(* Logix 5000 project; controller APM Emulate 5570 rev 30.12; software revision 30.00 *)

TASK MainTask (continuous, watchdog 500 ms) : MainProgram

MODULES
   Local : Emulate 5570 (ICP 2, rev 30.12)
      I_O1 : vendor 1 type 0 code 15 (ICP 3, rev 1.1, Output RPI 150 ms)
      I_O2 : vendor 1 type 0 code 15 (ICP 4, rev 1.1, Output RPI 150 ms)
END_MODULES

VAR_GLOBAL   (* controller tags *)
   CT_AXIS_DIST : AXIS_VIRTUAL;
   MTN : MOTION_GROUP;
   PNT_AXIS_MTA : AXIS_VIRTUAL;
   PNT_AXIS_MTB : AXIS_VIRTUAL;
   PNT_AXIS_MTC : AXIS_VIRTUAL;
END_VAR

PROGRAM MainProgram   (* main routine MainRoutine *)
VAR
   CT_ACT_CT0 : BOOL;
   CT_ACT_CT1 : BOOL;
   CT_ACT_CT2 : BOOL;
   CT_ACT_CT3 : BOOL;
   CT_ACT_CT4 : BOOL;
   CT_ACT_CT5 : BOOL;
   CT_ACT_CT6 : BOOL;
   CT_ACT_HOM0 : BOOL;
   CT_ACT_HOM1 : BOOL;
   CT_ACT_HOM2 : BOOL;
   CT_ACT_HOM3 : BOOL;
   CT_ACT_STP : BOOL;
   CT_AXIS_CT1 : MOTION_INSTRUCTION;
   CT_AXIS_CT4 : MOTION_INSTRUCTION;
   CT_AXIS_HOM0 : MOTION_INSTRUCTION;
   CT_AXIS_HOM1 : MOTION_INSTRUCTION;
   CT_AXIS_HOM2 : MOTION_INSTRUCTION;
   CT_CA_AVC : BOOL;
   CT_CA_RET : BOOL;
   CT_CC_AVC : BOOL;
   CT_CC_RET : BOOL;
   CT_CNT1 : COUNTER := (PRE := 18);
   CT_CP_AVC : BOOL;
   CT_CP_RET : BOOL;
   CT_DIST : INT;
   CT_ISOVER : BOOL;
   CT_MASD_DIST : MOTION_INSTRUCTION;
   CT_MASR_DIST : MOTION_INSTRUCTION;
   CT_OK : BOOL;
   CT_PBT_ESTP : ALIAS FOR Local:4:I.Data[1].0;
   CT_PBT_HOM : ALIAS FOR Local:4:I.Data[1].2;
   CT_PBT_STA : ALIAS FOR Local:4:I.Data[1].1;
   CT_SEN_CaAvc : ALIAS FOR Local:4:I.Data[1].4;
   CT_SEN_CaRet : ALIAS FOR Local:4:I.Data[1].3;
   CT_SEN_CcAvc : ALIAS FOR Local:4:I.Data[1].6;
   CT_SEN_CcRet : ALIAS FOR Local:4:I.Data[1].5;
   CT_SEN_CpAvc : ALIAS FOR Local:4:I.Data[1].8;
   CT_SEN_CpRet : ALIAS FOR Local:4:I.Data[1].7;
   CT_SEN_MAT : ALIAS FOR Local:4:I.Data[1].9;
   MAIN_ACTIVE : BOOL;
   MAIN_PBT_ESTP : ALIAS FOR Local:3:I.Data[1].0;
   MAIN_PBT_STA : ALIAS FOR Local:3:I.Data[1].1;
   PNT_ACT1_MTA_MAM : MOTION_INSTRUCTION;
   PNT_ACT1_MTB_MAM : MOTION_INSTRUCTION;
   PNT_ACT2_MTC_MAM : MOTION_INSTRUCTION;
   PNT_ACT3_MTA_MAM : MOTION_INSTRUCTION;
   PNT_ACT3_MTB_MAM : MOTION_INSTRUCTION;
   PNT_ACT_0 : BOOL;
   PNT_ACT_1 : BOOL;
   PNT_ACT_2 : BOOL;
   PNT_ACT_3 : BOOL;
   PNT_ACT_4 : BOOL;
   PNT_ACT_HOM : BOOL;
   PNT_ACTH_MTA_MAM : MOTION_INSTRUCTION;
   PNT_ACTH_MTB_MAM : MOTION_INSTRUCTION;
   PNT_ACTH_MTC_MAM : MOTION_INSTRUCTION;
   PNT_CNT1 : COUNTER := (PRE := 3);
   PNT_ISHOM : BOOL;
   PNT_ISOVER : BOOL;
   PNT_MASD_MTA : MOTION_INSTRUCTION;
   PNT_MASD_MTB : MOTION_INSTRUCTION;
   PNT_MASD_MTC : MOTION_INSTRUCTION;
   PNT_MASR_MTA : MOTION_INSTRUCTION;
   PNT_MASR_MTB : MOTION_INSTRUCTION;
   PNT_MASR_MTC : MOTION_INSTRUCTION;
   PNT_MTA_AVC : BOOL;
   PNT_MTA_RET : BOOL;
   PNT_MTA_STP : BOOL;
   PNT_MTB_AVC : BOOL;
   PNT_MTB_RET : BOOL;
   PNT_MTB_STP : BOOL;
   PNT_MTC_AVC : BOOL;
   PNT_MTC_RET : BOOL;
   PNT_MTC_STP : BOOL;
   PNT_PBT_HOM : ALIAS FOR Local:3:I.Data[1].10;
   PNT_PBT_STA : ALIAS FOR Local:3:I.Data[1].11;
   PNT_PBT_STP : ALIAS FOR Local:3:I.Data[1].12;
   PNT_SEN_1 : ALIAS FOR Local:3:I.Data[1].13;
   PNT_SEN_2 : ALIAS FOR Local:3:I.Data[1].14;
   PNT_SEN_3 : ALIAS FOR Local:3:I.Data[1].15;
   PNT_SEN_4 : ALIAS FOR Local:3:I.Data[1].16;
   PNT_SEN_5 : ALIAS FOR Local:3:I.Data[1].17;
   PNT_SEN_6 : ALIAS FOR Local:3:I.Data[1].18;
   PNT_SEN_7 : ALIAS FOR Local:3:I.Data[1].19;
   PNT_TM1 : TIMER := (PRE := 2000);
END_VAR

ROUTINE Corte_actions   (* ladder *)
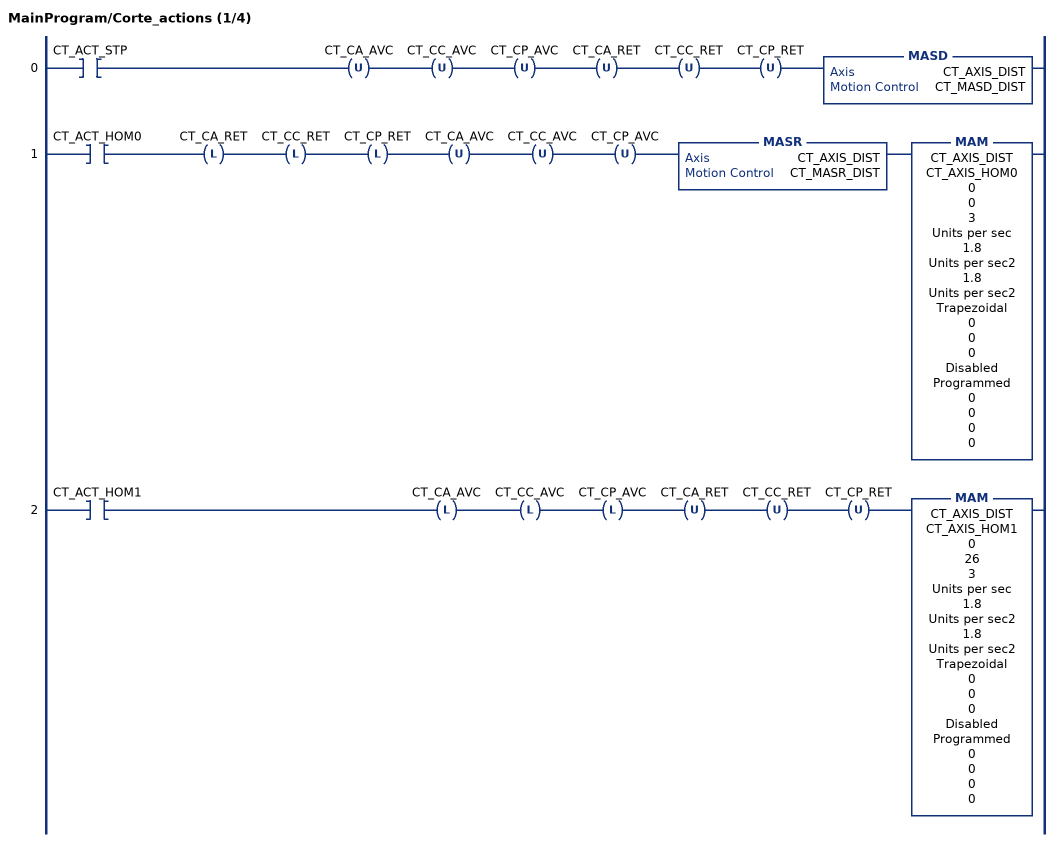
   0: XIC(CT_ACT_STP)OTU(CT_CA_AVC)OTU(CT_CC_AVC)OTU(CT_CP_AVC)OTU(CT_CA_RET)OTU(CT_CC_RET)OTU(CT_CP_RET)MASD(CT_AXIS_DIST,CT_MASD_DIST);
   1: XIC(CT_ACT_HOM0)OTL(CT_CA_RET)OTL(CT_CC_RET)OTL(CT_CP_RET)OTU(CT_CA_AVC)OTU(CT_CC_AVC)OTU(CT_CP_AVC)MASR(CT_AXIS_DIST,CT_MASR_DIST)MAM(CT_AXIS_DIST,CT_AXIS_HOM0,0,0,3,Units per sec,1.8,Units per sec2,1.8,Units per sec2,Trapezoidal,0,0,0,Disabled,Programmed,0,0,0,0);
   2: XIC(CT_ACT_HOM1)OTL(CT_CA_AVC)OTL(CT_CC_AVC)OTL(CT_CP_AVC)OTU(CT_CA_RET)OTU(CT_CC_RET)OTU(CT_CP_RET)MAM(CT_AXIS_DIST,CT_AXIS_HOM1,0,26,3,Units per sec,1.8,Units per sec2,1.8,Units per sec2,Trapezoidal,0,0,0,Disabled,Programmed,0,0,0,0);
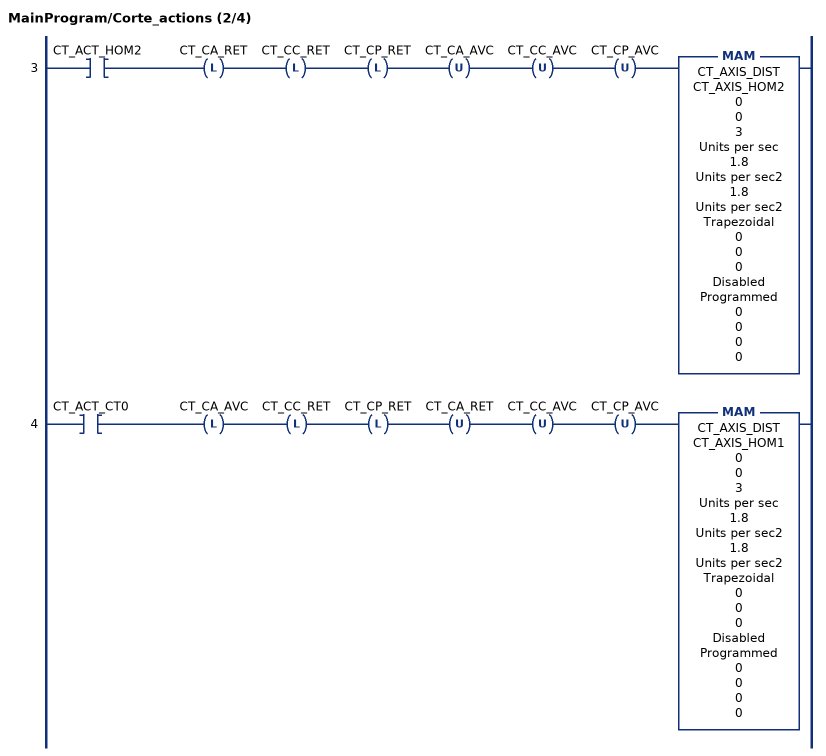
   3: XIC(CT_ACT_HOM2)OTL(CT_CA_RET)OTL(CT_CC_RET)OTL(CT_CP_RET)OTU(CT_CA_AVC)OTU(CT_CC_AVC)OTU(CT_CP_AVC)MAM(CT_AXIS_DIST,CT_AXIS_HOM2,0,0,3,Units per sec,1.8,Units per sec2,1.8,Units per sec2,Trapezoidal,0,0,0,Disabled,Programmed,0,0,0,0);
   4: XIC(CT_ACT_CT0)OTL(CT_CA_AVC)OTL(CT_CC_RET)OTL(CT_CP_RET)OTU(CT_CA_RET)OTU(CT_CC_AVC)OTU(CT_CP_AVC)MAM(CT_AXIS_DIST,CT_AXIS_HOM1,0,0,3,Units per sec,1.8,Units per sec2,1.8,Units per sec2,Trapezoidal,0,0,0,Disabled,Programmed,0,0,0,0);
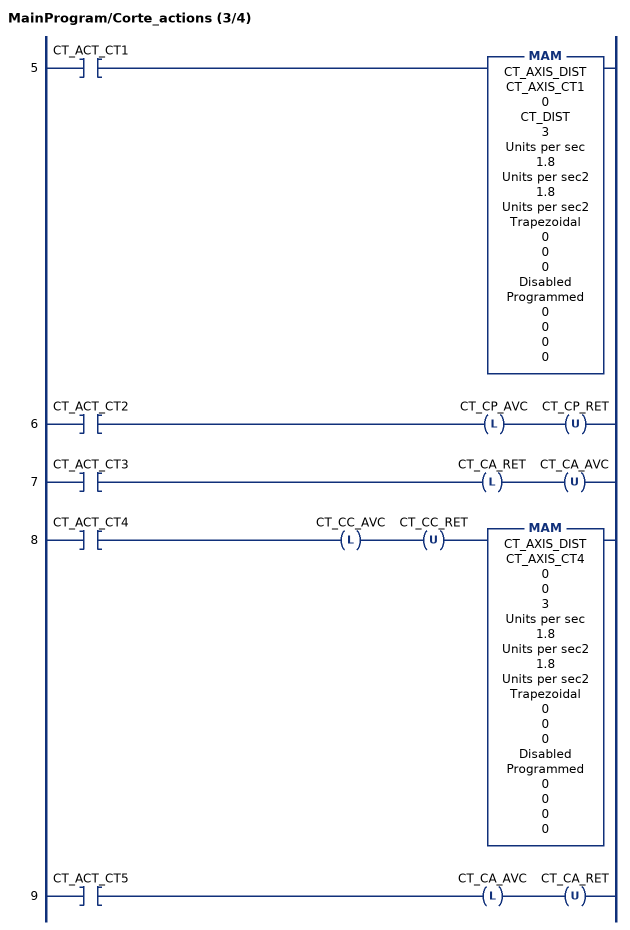
   5: XIC(CT_ACT_CT1)MAM(CT_AXIS_DIST,CT_AXIS_CT1,0,CT_DIST,3,Units per sec,1.8,Units per sec2,1.8,Units per sec2,Trapezoidal,0,0,0,Disabled,Programmed,0,0,0,0);
   6: XIC(CT_ACT_CT2)OTL(CT_CP_AVC)OTU(CT_CP_RET);
   7: XIC(CT_ACT_CT3)OTL(CT_CA_RET)OTU(CT_CA_AVC);
   8: XIC(CT_ACT_CT4)OTL(CT_CC_AVC)OTU(CT_CC_RET)MAM(CT_AXIS_DIST,CT_AXIS_CT4,0,0,3,Units per sec,1.8,Units per sec2,1.8,Units per sec2,Trapezoidal,0,0,0,Disabled,Programmed,0,0,0,0);
   9: XIC(CT_ACT_CT5)OTL(CT_CA_AVC)OTU(CT_CA_RET);
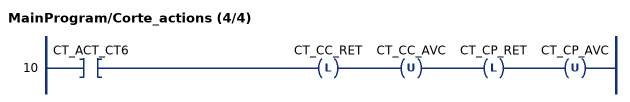
   10: XIC(CT_ACT_CT6)OTL(CT_CC_RET)OTU(CT_CC_AVC)OTL(CT_CP_RET)OTU(CT_CP_AVC);
END_ROUTINE

ROUTINE Corte_logic   (* ladder *)
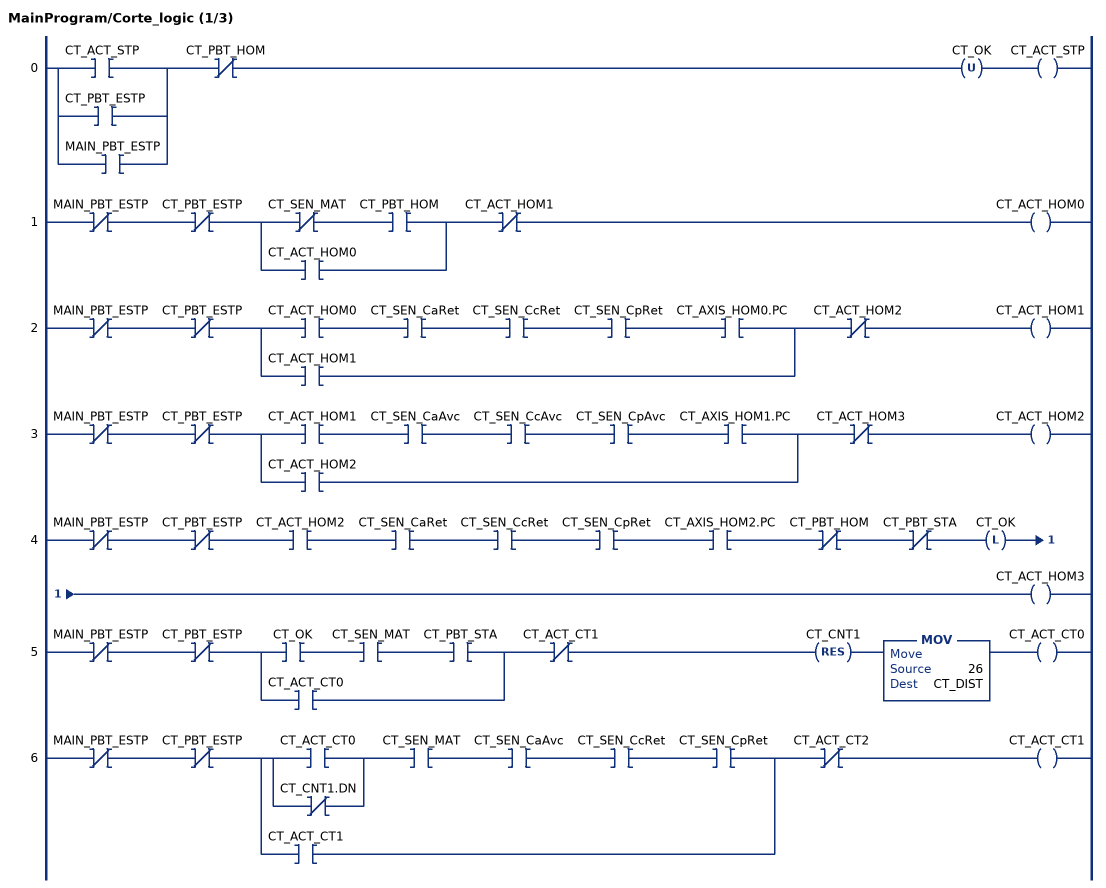
   0: [XIC(CT_ACT_STP) ,XIC(CT_PBT_ESTP) ,XIC(MAIN_PBT_ESTP) ]XIO(CT_PBT_HOM)OTU(CT_OK)OTE(CT_ACT_STP);
   1: XIO(MAIN_PBT_ESTP)XIO(CT_PBT_ESTP)[XIO(CT_SEN_MAT) XIC(CT_PBT_HOM) ,XIC(CT_ACT_HOM0) ]XIO(CT_ACT_HOM1)OTE(CT_ACT_HOM0);
   2: XIO(MAIN_PBT_ESTP)XIO(CT_PBT_ESTP)[XIC(CT_ACT_HOM0) XIC(CT_SEN_CaRet) XIC(CT_SEN_CcRet) XIC(CT_SEN_CpRet) XIC(CT_AXIS_HOM0.PC) ,XIC(CT_ACT_HOM1) ]XIO(CT_ACT_HOM2)OTE(CT_ACT_HOM1);
   3: XIO(MAIN_PBT_ESTP)XIO(CT_PBT_ESTP)[XIC(CT_ACT_HOM1) XIC(CT_SEN_CaAvc) XIC(CT_SEN_CcAvc) XIC(CT_SEN_CpAvc) XIC(CT_AXIS_HOM1.PC) ,XIC(CT_ACT_HOM2) ]XIO(CT_ACT_HOM3)OTE(CT_ACT_HOM2);
   4: XIO(MAIN_PBT_ESTP)XIO(CT_PBT_ESTP)XIC(CT_ACT_HOM2)XIC(CT_SEN_CaRet)XIC(CT_SEN_CcRet)XIC(CT_SEN_CpRet)XIC(CT_AXIS_HOM2.PC)XIO(CT_PBT_HOM)XIO(CT_PBT_STA)OTL(CT_OK)OTE(CT_ACT_HOM3);
   5: XIO(MAIN_PBT_ESTP)XIO(CT_PBT_ESTP)[XIC(CT_OK) XIC(CT_SEN_MAT) XIC(CT_PBT_STA) ,XIC(CT_ACT_CT0) ]XIO(CT_ACT_CT1)RES(CT_CNT1)MOV(26,CT_DIST)OTE(CT_ACT_CT0);
   6: XIO(MAIN_PBT_ESTP)XIO(CT_PBT_ESTP)[[XIC(CT_ACT_CT0) ,XIO(CT_CNT1.DN) ] XIC(CT_SEN_MAT) XIC(CT_SEN_CaAvc) XIC(CT_SEN_CcRet) XIC(CT_SEN_CpRet) ,XIC(CT_ACT_CT1) ]XIO(CT_ACT_CT2)OTE(CT_ACT_CT1);
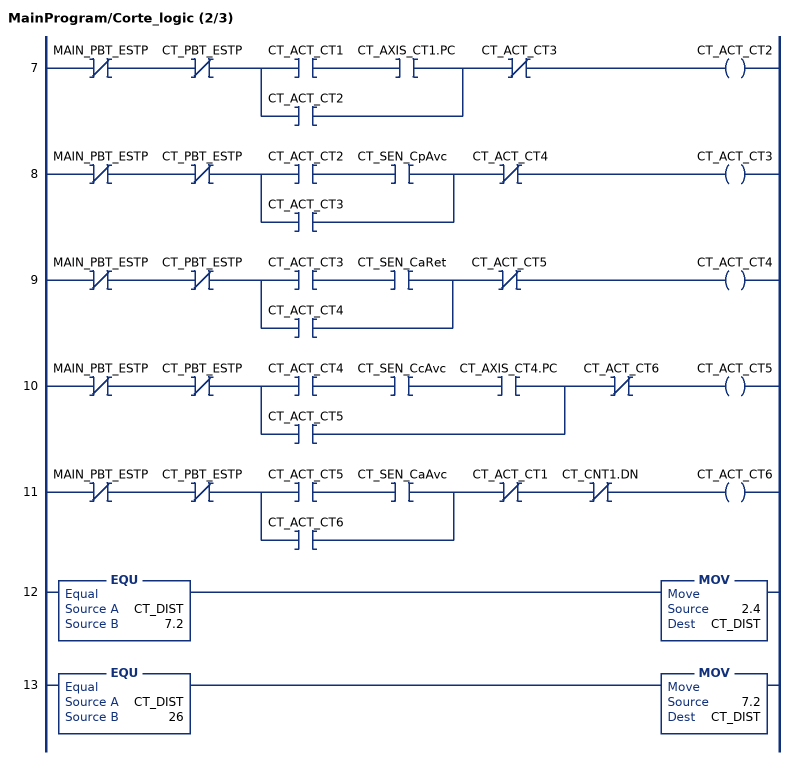
   7: XIO(MAIN_PBT_ESTP)XIO(CT_PBT_ESTP)[XIC(CT_ACT_CT1) XIC(CT_AXIS_CT1.PC) ,XIC(CT_ACT_CT2) ]XIO(CT_ACT_CT3)OTE(CT_ACT_CT2);
   8: XIO(MAIN_PBT_ESTP)XIO(CT_PBT_ESTP)[XIC(CT_ACT_CT2) XIC(CT_SEN_CpAvc) ,XIC(CT_ACT_CT3) ]XIO(CT_ACT_CT4)OTE(CT_ACT_CT3);
   9: XIO(MAIN_PBT_ESTP)XIO(CT_PBT_ESTP)[XIC(CT_ACT_CT3) XIC(CT_SEN_CaRet) ,XIC(CT_ACT_CT4) ]XIO(CT_ACT_CT5)OTE(CT_ACT_CT4);
   10: XIO(MAIN_PBT_ESTP)XIO(CT_PBT_ESTP)[XIC(CT_ACT_CT4) XIC(CT_SEN_CcAvc) XIC(CT_AXIS_CT4.PC) ,XIC(CT_ACT_CT5) ]XIO(CT_ACT_CT6)OTE(CT_ACT_CT5);
   11: XIO(MAIN_PBT_ESTP)XIO(CT_PBT_ESTP)[XIC(CT_ACT_CT5) XIC(CT_SEN_CaAvc) ,XIC(CT_ACT_CT6) ]XIO(CT_ACT_CT1)XIO(CT_CNT1.DN)OTE(CT_ACT_CT6);
   12: EQU(CT_DIST,7.2)MOV(2.4,CT_DIST);
   13: EQU(CT_DIST,26)MOV(7.2,CT_DIST);
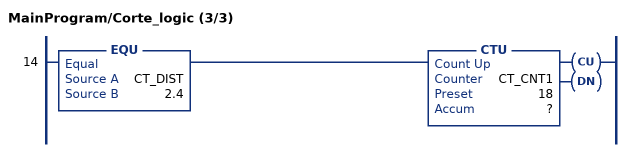
   14: EQU(CT_DIST,2.4)CTU(CT_CNT1,?,?);
END_ROUTINE

ROUTINE MainRoutine   (* ladder *)
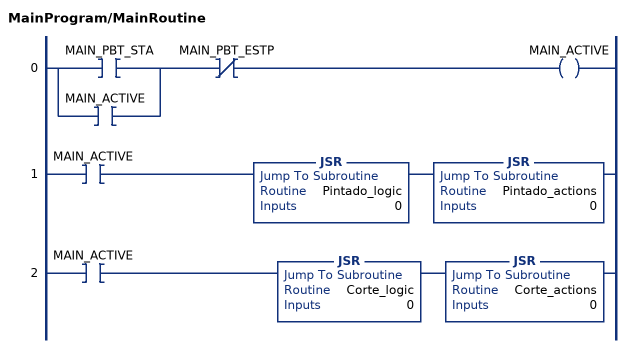
   0: [XIC(MAIN_PBT_STA) ,XIC(MAIN_ACTIVE) ]XIO(MAIN_PBT_ESTP)OTE(MAIN_ACTIVE);
   1: XIC(MAIN_ACTIVE)JSR(Pintado_logic,0)JSR(Pintado_actions,0);
   2: XIC(MAIN_ACTIVE)JSR(Corte_logic,0)JSR(Corte_actions,0);
END_ROUTINE

ROUTINE Pintado_actions   (* ladder *)
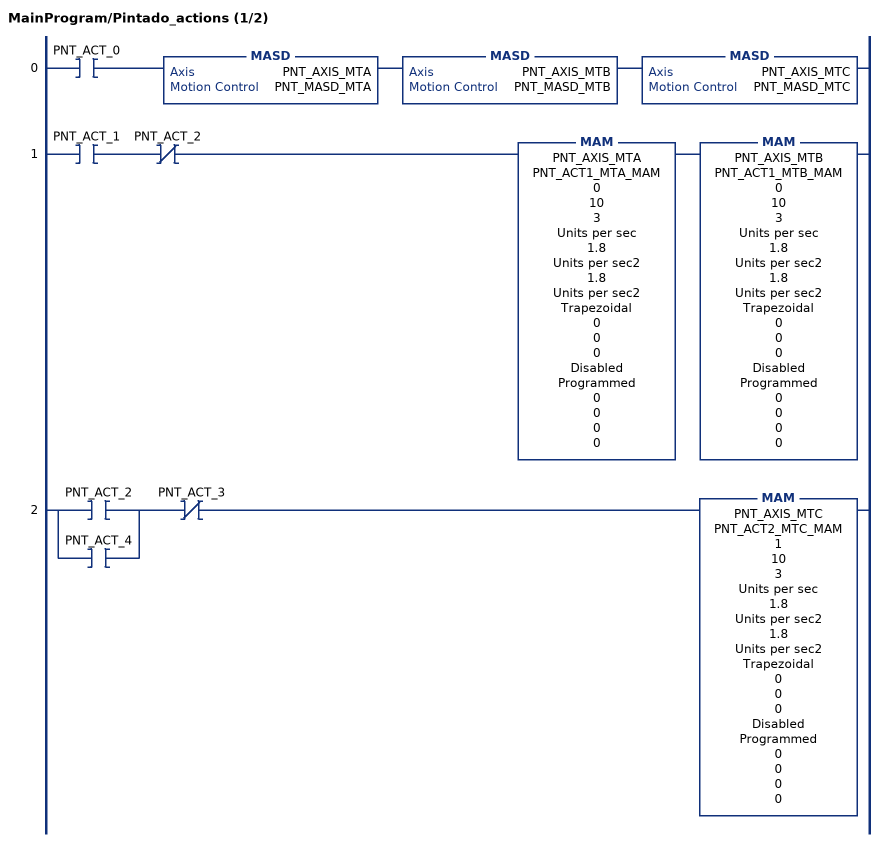
   0: XIC(PNT_ACT_0)MASD(PNT_AXIS_MTA,PNT_MASD_MTA)MASD(PNT_AXIS_MTB,PNT_MASD_MTB)MASD(PNT_AXIS_MTC,PNT_MASD_MTC);
   1: XIC(PNT_ACT_1)XIO(PNT_ACT_2)MAM(PNT_AXIS_MTA,PNT_ACT1_MTA_MAM,0,10,3,Units per sec,1.8,Units per sec2,1.8,Units per sec2,Trapezoidal,0,0,0,Disabled,Programmed,0,0,0,0)MAM(PNT_AXIS_MTB,PNT_ACT1_MTB_MAM,0,10,3,Units per sec,1.8,Units per sec2,1.8,Units per sec2,Trapezoidal,0,0,0,Disabled,Programmed,0,0,0,0);
   2: [XIC(PNT_ACT_2) ,XIC(PNT_ACT_4) ]XIO(PNT_ACT_3)MAM(PNT_AXIS_MTC,PNT_ACT2_MTC_MAM,1,10,3,Units per sec,1.8,Units per sec2,1.8,Units per sec2,Trapezoidal,0,0,0,Disabled,Programmed,0,0,0,0);
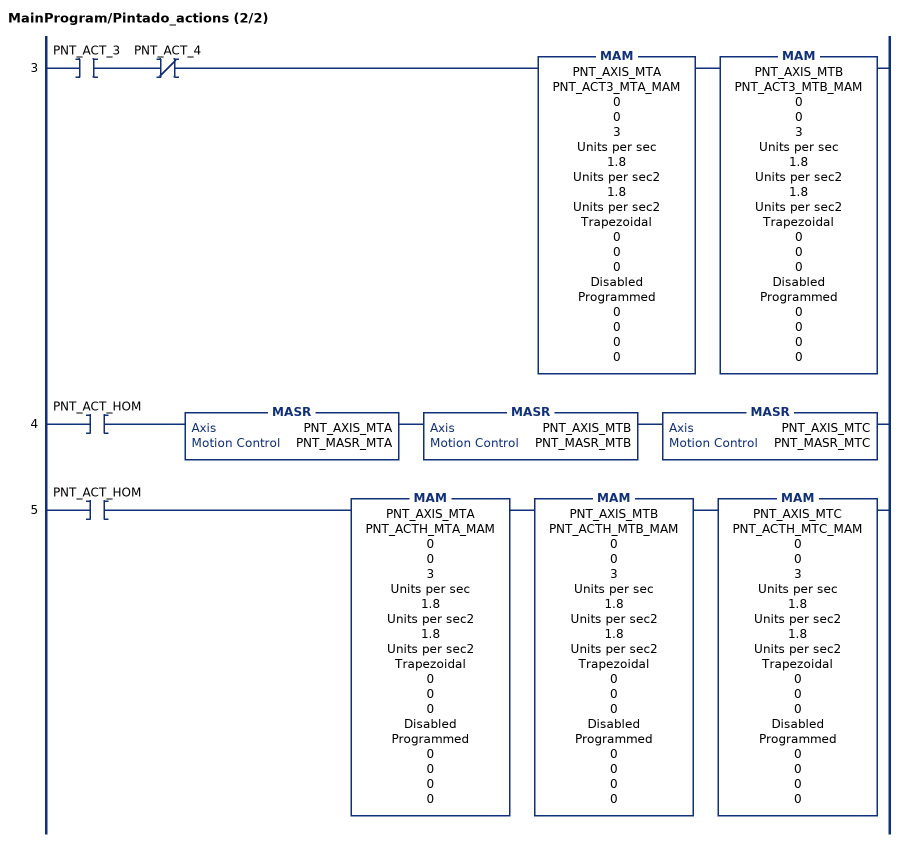
   3: XIC(PNT_ACT_3)XIO(PNT_ACT_4)MAM(PNT_AXIS_MTA,PNT_ACT3_MTA_MAM,0,0,3,Units per sec,1.8,Units per sec2,1.8,Units per sec2,Trapezoidal,0,0,0,Disabled,Programmed,0,0,0,0)MAM(PNT_AXIS_MTB,PNT_ACT3_MTB_MAM,0,0,3,Units per sec,1.8,Units per sec2,1.8,Units per sec2,Trapezoidal,0,0,0,Disabled,Programmed,0,0,0,0);
   4: XIC(PNT_ACT_HOM)MASR(PNT_AXIS_MTA,PNT_MASR_MTA)MASR(PNT_AXIS_MTB,PNT_MASR_MTB)MASR(PNT_AXIS_MTC,PNT_MASR_MTC);
   5: XIC(PNT_ACT_HOM)MAM(PNT_AXIS_MTA,PNT_ACTH_MTA_MAM,0,0,3,Units per sec,1.8,Units per sec2,1.8,Units per sec2,Trapezoidal,0,0,0,Disabled,Programmed,0,0,0,0)MAM(PNT_AXIS_MTB,PNT_ACTH_MTB_MAM,0,0,3,Units per sec,1.8,Units per sec2,1.8,Units per sec2,Trapezoidal,0,0,0,Disabled,Programmed,0,0,0,0)MAM(PNT_AXIS_MTC,PNT_ACTH_MTC_MAM,0,0,3,Units per sec,1.8,Units per sec2,1.8,Units per sec2,Trapezoidal,0,0,0,Disabled,Programmed,0,0,0,0);
END_ROUTINE

ROUTINE Pintado_logic   (* ladder *)
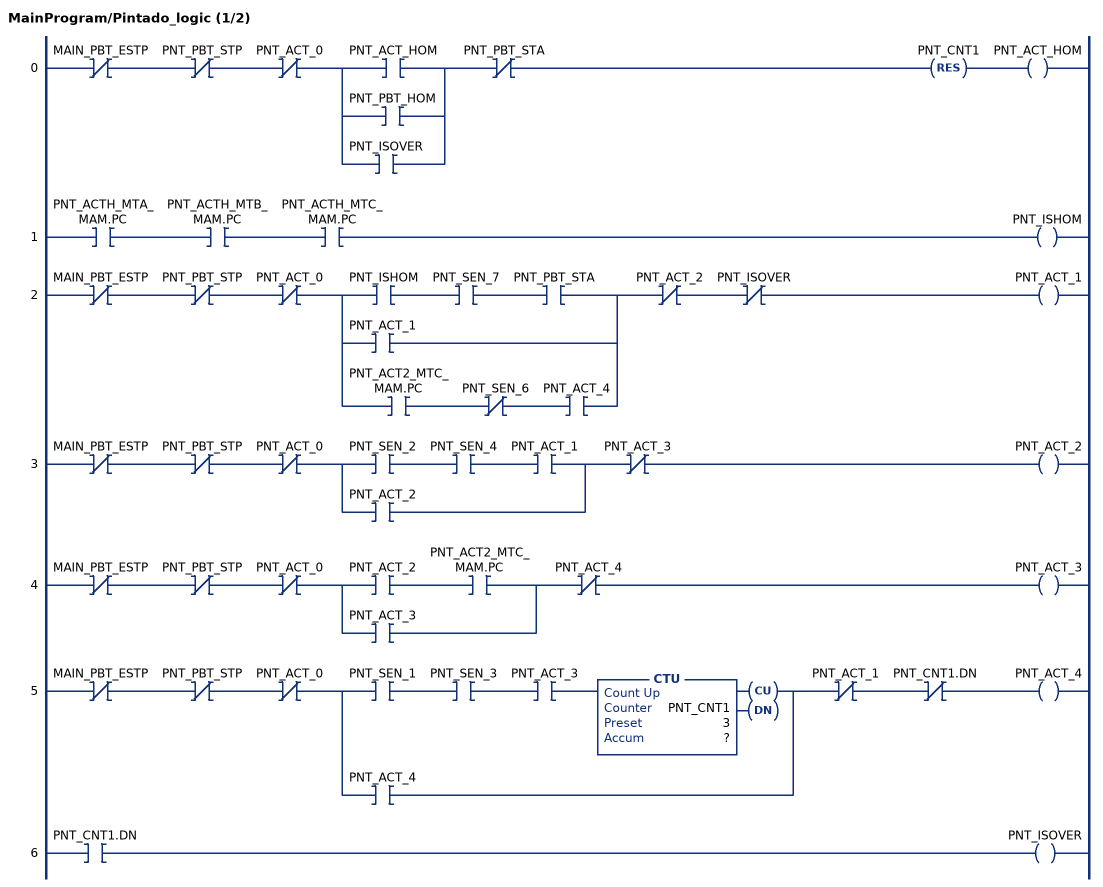
   0: XIO(MAIN_PBT_ESTP)XIO(PNT_PBT_STP)XIO(PNT_ACT_0)[XIC(PNT_ACT_HOM) ,XIC(PNT_PBT_HOM) ,XIC(PNT_ISOVER) ]XIO(PNT_PBT_STA)RES(PNT_CNT1)OTE(PNT_ACT_HOM);
   1: XIC(PNT_ACTH_MTA_MAM.PC)XIC(PNT_ACTH_MTB_MAM.PC)XIC(PNT_ACTH_MTC_MAM.PC)OTE(PNT_ISHOM);
   2: XIO(MAIN_PBT_ESTP)XIO(PNT_PBT_STP)XIO(PNT_ACT_0)[XIC(PNT_ISHOM) XIC(PNT_SEN_7) XIC(PNT_PBT_STA) ,XIC(PNT_ACT_1) ,XIC(PNT_ACT2_MTC_MAM.PC) XIO(PNT_SEN_6) XIC(PNT_ACT_4) ]XIO(PNT_ACT_2)XIO(PNT_ISOVER)OTE(PNT_ACT_1);
   3: XIO(MAIN_PBT_ESTP)XIO(PNT_PBT_STP)XIO(PNT_ACT_0)[XIC(PNT_SEN_2) XIC(PNT_SEN_4) XIC(PNT_ACT_1) ,XIC(PNT_ACT_2) ]XIO(PNT_ACT_3)OTE(PNT_ACT_2);
   4: XIO(MAIN_PBT_ESTP)XIO(PNT_PBT_STP)XIO(PNT_ACT_0)[XIC(PNT_ACT_2) XIC(PNT_ACT2_MTC_MAM.PC) ,XIC(PNT_ACT_3) ]XIO(PNT_ACT_4)OTE(PNT_ACT_3);
   5: XIO(MAIN_PBT_ESTP)XIO(PNT_PBT_STP)XIO(PNT_ACT_0)[XIC(PNT_SEN_1) XIC(PNT_SEN_3) XIC(PNT_ACT_3) CTU(PNT_CNT1,?,?) ,XIC(PNT_ACT_4) ]XIO(PNT_ACT_1)XIO(PNT_CNT1.DN)OTE(PNT_ACT_4);
   6: XIC(PNT_CNT1.DN)OTE(PNT_ISOVER);
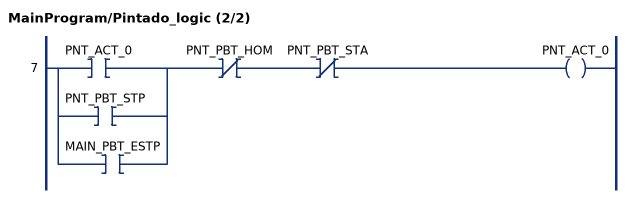
   7: [XIC(PNT_ACT_0) ,XIC(PNT_PBT_STP) ,XIC(MAIN_PBT_ESTP) ]XIO(PNT_PBT_HOM)XIO(PNT_PBT_STA)OTE(PNT_ACT_0);
END_ROUTINE

ROUTINE temp   (* ladder *)
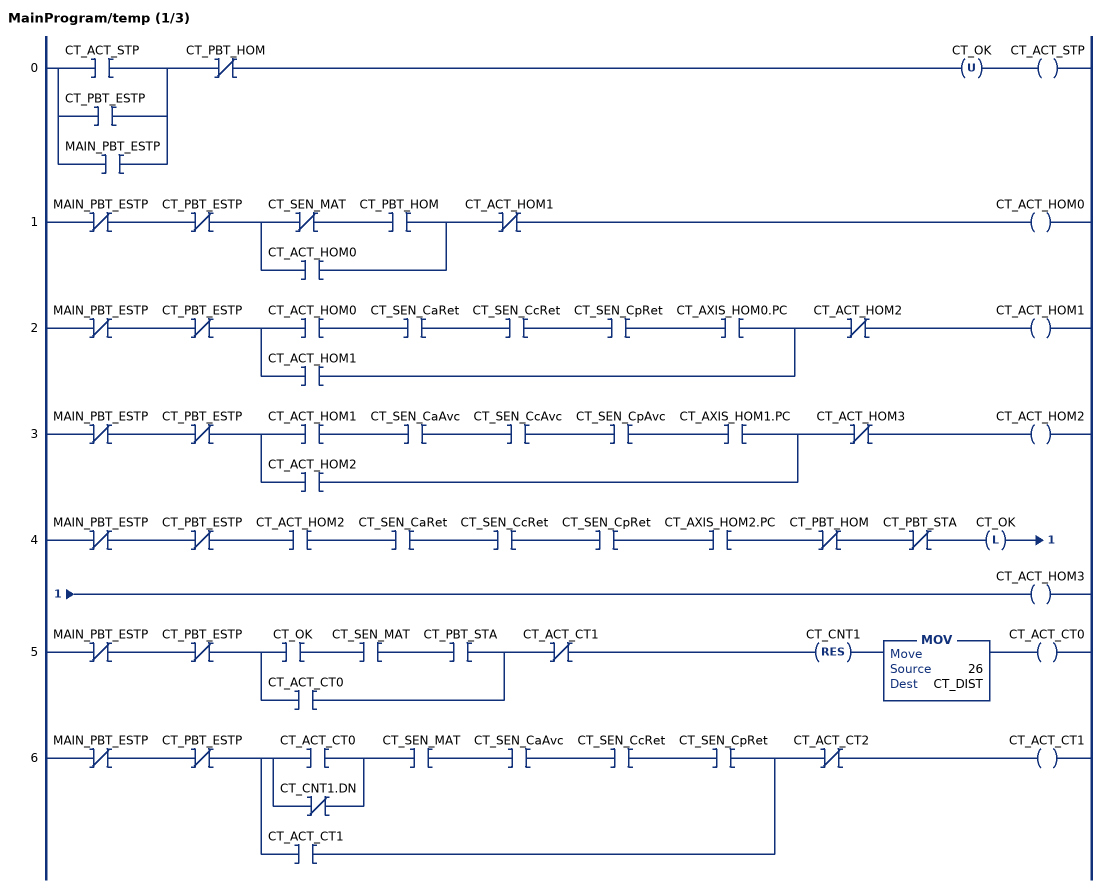
   0: [XIC(CT_ACT_STP) ,XIC(CT_PBT_ESTP) ,XIC(MAIN_PBT_ESTP) ]XIO(CT_PBT_HOM)OTU(CT_OK)OTE(CT_ACT_STP);
   1: XIO(MAIN_PBT_ESTP)XIO(CT_PBT_ESTP)[XIO(CT_SEN_MAT) XIC(CT_PBT_HOM) ,XIC(CT_ACT_HOM0) ]XIO(CT_ACT_HOM1)OTE(CT_ACT_HOM0);
   2: XIO(MAIN_PBT_ESTP)XIO(CT_PBT_ESTP)[XIC(CT_ACT_HOM0) XIC(CT_SEN_CaRet) XIC(CT_SEN_CcRet) XIC(CT_SEN_CpRet) XIC(CT_AXIS_HOM0.PC) ,XIC(CT_ACT_HOM1) ]XIO(CT_ACT_HOM2)OTE(CT_ACT_HOM1);
   3: XIO(MAIN_PBT_ESTP)XIO(CT_PBT_ESTP)[XIC(CT_ACT_HOM1) XIC(CT_SEN_CaAvc) XIC(CT_SEN_CcAvc) XIC(CT_SEN_CpAvc) XIC(CT_AXIS_HOM1.PC) ,XIC(CT_ACT_HOM2) ]XIO(CT_ACT_HOM3)OTE(CT_ACT_HOM2);
   4: XIO(MAIN_PBT_ESTP)XIO(CT_PBT_ESTP)XIC(CT_ACT_HOM2)XIC(CT_SEN_CaRet)XIC(CT_SEN_CcRet)XIC(CT_SEN_CpRet)XIC(CT_AXIS_HOM2.PC)XIO(CT_PBT_HOM)XIO(CT_PBT_STA)OTL(CT_OK)OTE(CT_ACT_HOM3);
   5: XIO(MAIN_PBT_ESTP)XIO(CT_PBT_ESTP)[XIC(CT_OK) XIC(CT_SEN_MAT) XIC(CT_PBT_STA) ,XIC(CT_ACT_CT0) ]XIO(CT_ACT_CT1)RES(CT_CNT1)MOV(26,CT_DIST)OTE(CT_ACT_CT0);
   6: XIO(MAIN_PBT_ESTP)XIO(CT_PBT_ESTP)[[XIC(CT_ACT_CT0) ,XIO(CT_CNT1.DN) ] XIC(CT_SEN_MAT) XIC(CT_SEN_CaAvc) XIC(CT_SEN_CcRet) XIC(CT_SEN_CpRet) ,XIC(CT_ACT_CT1) ]XIO(CT_ACT_CT2)OTE(CT_ACT_CT1);
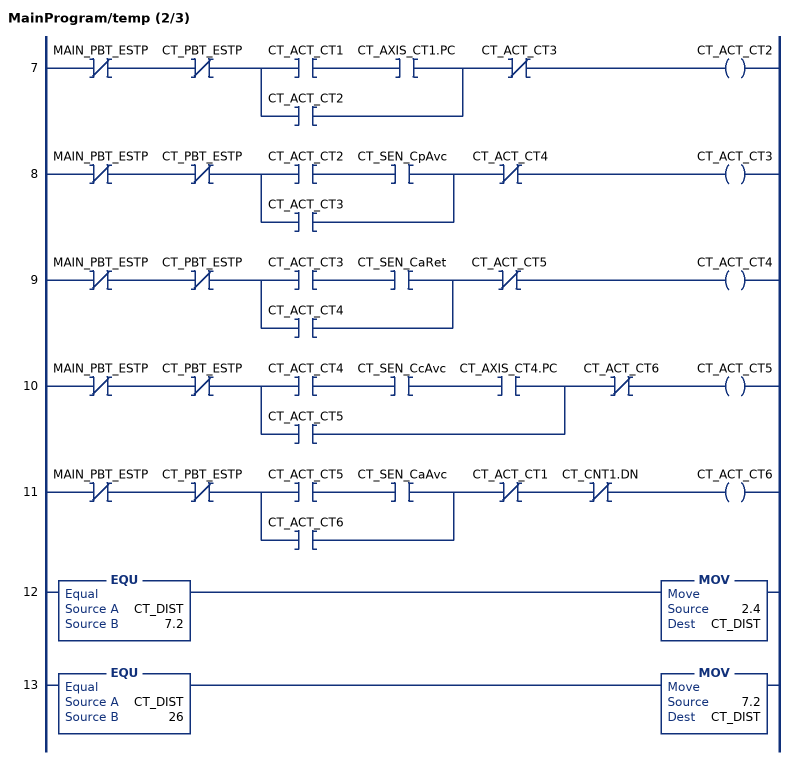
   7: XIO(MAIN_PBT_ESTP)XIO(CT_PBT_ESTP)[XIC(CT_ACT_CT1) XIC(CT_AXIS_CT1.PC) ,XIC(CT_ACT_CT2) ]XIO(CT_ACT_CT3)OTE(CT_ACT_CT2);
   8: XIO(MAIN_PBT_ESTP)XIO(CT_PBT_ESTP)[XIC(CT_ACT_CT2) XIC(CT_SEN_CpAvc) ,XIC(CT_ACT_CT3) ]XIO(CT_ACT_CT4)OTE(CT_ACT_CT3);
   9: XIO(MAIN_PBT_ESTP)XIO(CT_PBT_ESTP)[XIC(CT_ACT_CT3) XIC(CT_SEN_CaRet) ,XIC(CT_ACT_CT4) ]XIO(CT_ACT_CT5)OTE(CT_ACT_CT4);
   10: XIO(MAIN_PBT_ESTP)XIO(CT_PBT_ESTP)[XIC(CT_ACT_CT4) XIC(CT_SEN_CcAvc) XIC(CT_AXIS_CT4.PC) ,XIC(CT_ACT_CT5) ]XIO(CT_ACT_CT6)OTE(CT_ACT_CT5);
   11: XIO(MAIN_PBT_ESTP)XIO(CT_PBT_ESTP)[XIC(CT_ACT_CT5) XIC(CT_SEN_CaAvc) ,XIC(CT_ACT_CT6) ]XIO(CT_ACT_CT1)XIO(CT_CNT1.DN)OTE(CT_ACT_CT6);
   12: EQU(CT_DIST,7.2)MOV(2.4,CT_DIST);
   13: EQU(CT_DIST,26)MOV(7.2,CT_DIST);
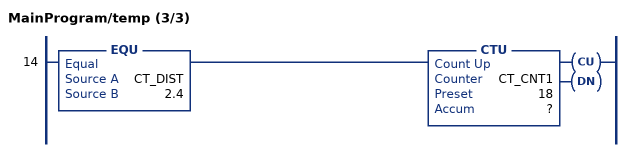
   14: EQU(CT_DIST,2.4)CTU(CT_CNT1,?,?);
END_ROUTINE

ROUTINE tempact   (* ladder *)
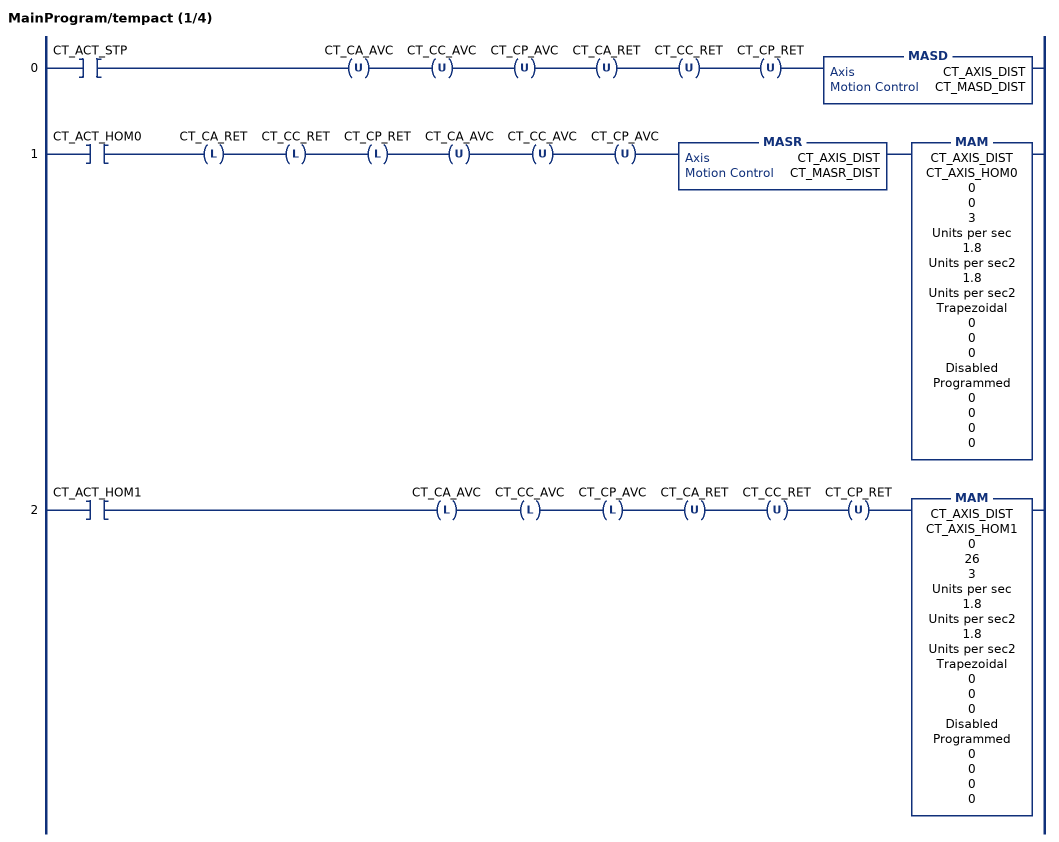
   0: XIC(CT_ACT_STP)OTU(CT_CA_AVC)OTU(CT_CC_AVC)OTU(CT_CP_AVC)OTU(CT_CA_RET)OTU(CT_CC_RET)OTU(CT_CP_RET)MASD(CT_AXIS_DIST,CT_MASD_DIST);
   1: XIC(CT_ACT_HOM0)OTL(CT_CA_RET)OTL(CT_CC_RET)OTL(CT_CP_RET)OTU(CT_CA_AVC)OTU(CT_CC_AVC)OTU(CT_CP_AVC)MASR(CT_AXIS_DIST,CT_MASR_DIST)MAM(CT_AXIS_DIST,CT_AXIS_HOM0,0,0,3,Units per sec,1.8,Units per sec2,1.8,Units per sec2,Trapezoidal,0,0,0,Disabled,Programmed,0,0,0,0);
   2: XIC(CT_ACT_HOM1)OTL(CT_CA_AVC)OTL(CT_CC_AVC)OTL(CT_CP_AVC)OTU(CT_CA_RET)OTU(CT_CC_RET)OTU(CT_CP_RET)MAM(CT_AXIS_DIST,CT_AXIS_HOM1,0,26,3,Units per sec,1.8,Units per sec2,1.8,Units per sec2,Trapezoidal,0,0,0,Disabled,Programmed,0,0,0,0);
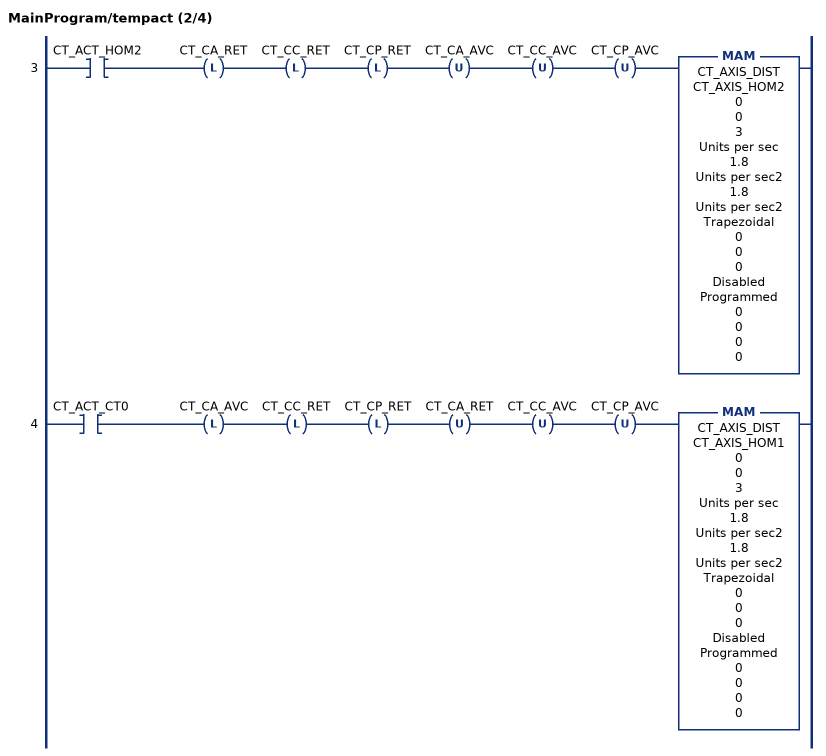
   3: XIC(CT_ACT_HOM2)OTL(CT_CA_RET)OTL(CT_CC_RET)OTL(CT_CP_RET)OTU(CT_CA_AVC)OTU(CT_CC_AVC)OTU(CT_CP_AVC)MAM(CT_AXIS_DIST,CT_AXIS_HOM2,0,0,3,Units per sec,1.8,Units per sec2,1.8,Units per sec2,Trapezoidal,0,0,0,Disabled,Programmed,0,0,0,0);
   4: XIC(CT_ACT_CT0)OTL(CT_CA_AVC)OTL(CT_CC_RET)OTL(CT_CP_RET)OTU(CT_CA_RET)OTU(CT_CC_AVC)OTU(CT_CP_AVC)MAM(CT_AXIS_DIST,CT_AXIS_HOM1,0,0,3,Units per sec,1.8,Units per sec2,1.8,Units per sec2,Trapezoidal,0,0,0,Disabled,Programmed,0,0,0,0);
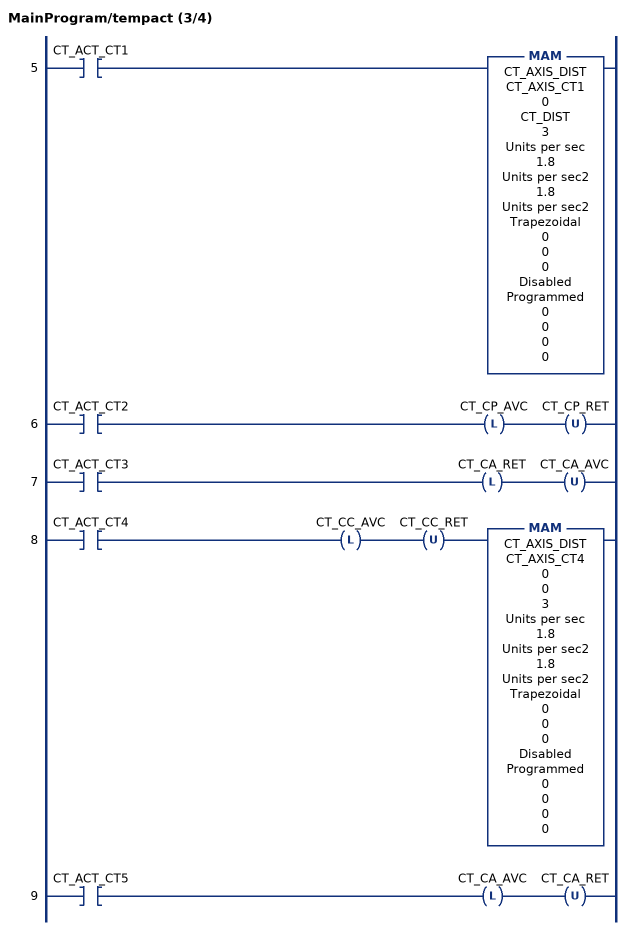
   5: XIC(CT_ACT_CT1)MAM(CT_AXIS_DIST,CT_AXIS_CT1,0,CT_DIST,3,Units per sec,1.8,Units per sec2,1.8,Units per sec2,Trapezoidal,0,0,0,Disabled,Programmed,0,0,0,0);
   6: XIC(CT_ACT_CT2)OTL(CT_CP_AVC)OTU(CT_CP_RET);
   7: XIC(CT_ACT_CT3)OTL(CT_CA_RET)OTU(CT_CA_AVC);
   8: XIC(CT_ACT_CT4)OTL(CT_CC_AVC)OTU(CT_CC_RET)MAM(CT_AXIS_DIST,CT_AXIS_CT4,0,0,3,Units per sec,1.8,Units per sec2,1.8,Units per sec2,Trapezoidal,0,0,0,Disabled,Programmed,0,0,0,0);
   9: XIC(CT_ACT_CT5)OTL(CT_CA_AVC)OTU(CT_CA_RET);
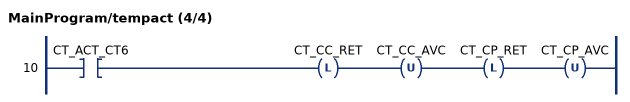
   10: XIC(CT_ACT_CT6)OTL(CT_CC_RET)OTU(CT_CC_AVC)OTL(CT_CP_RET)OTU(CT_CP_AVC);
END_ROUTINE
END_PROGRAM
